# EPICS substitutions: docs/example_ioc/IOCApp/Db/IOC.substitutions
file $(PICOHARP)/db/picoharp.db
{
pattern { DEVICE, PORT, CURRENT, EVENT_FAST, EVENT_5S, BUCKETS, BUCKETS_1, PROFILE }
    { "BL01B-DI-PICO-01", "PICO1", "SR-DI-DCCT-01:SIGNAL", "101", "102", "936", "935", "62" }
}
